PROGRAM P_PackML
VAR
	machine1	: Machine;
	eModeCommand: E_PMLProtectedUnitMode;
	eCommand	: E_PMLCommand;
END_VAR

machine1(
	eModeCommand	:= eModeCommand, 
	eCommand		:= eCommand, 
	eMode			=> , 
	eState			=> , 
	bUndefinedDone	=> , 
	bInvalidModeCommandOut=> , 
	bChangeIntoProduction=> );

END_PROGRAM

(* stored: Version 1.1.0.1
   POU P_PackML: Id {69c9c407-efe1-48a4-a030-598eddc6bb34}, SpecialFunc None *)
